// TIA Portal V17 export
// export: Created 2024-06-16T17:47:21.7318525Z, ExportSetting WithDefaults, DisplayName Totally Integrated Automation Portal, DisplayVersion V17, DisplayName TIA Portal Openness, DisplayVersion V17, DisplayName TIA Portal Version Control Interface, DisplayVersion V17, DisplayName STEP 7 Professional, DisplayVersion V17, DisplayName STEP 7 Safety, DisplayVersion V17, DisplayName WinCC Professional, DisplayVersion V17
DATA_BLOCK "S40_Acquitement"   // DB1050
VERSION : 0.1
// stored: AutoNumber false, DBAccessibleFromOPCUA true, DBAccessibleFromWebserver true, InstanceOfName S40_Acquitement_FB, InstanceOfType FB
"S40_Acquitement_FB"
   // VAR_OUTPUT
   //    "Step" : Int;
   // END_VAR
   // VAR
   //    Step_100 : Int;
   // END_VAR
BEGIN
END_DATA_BLOCK
